Staubli VAL3: copy_it.pgx

public program copy_it(string x_sCopy, string x_sPaste)
  local num i
begin
  // try to copy it
  if isDefined(tTraj[x_sCopy])
    // copy it
    tTraj[x_sPaste]=tTraj[x_sCopy]
    //
  endIf
end
